FUNCTION_BLOCK PlantProcess
  (* Standard: 61499-2 *)
  (* Version 0.1, 2017-00-02, hpea485, UOA *)
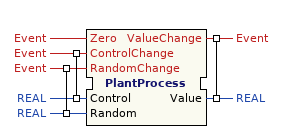
  EVENT_INPUT
    Zero;
    ControlChange WITH Control;
    RandomChange WITH Random;
  END_EVENT
  EVENT_OUTPUT
    ValueChange WITH Value;
  END_EVENT
  VAR_INPUT
    Control : REAL;
    Random : REAL := 0.0;
  END_VAR
  VAR_OUTPUT
    Value : REAL;
  END_VAR
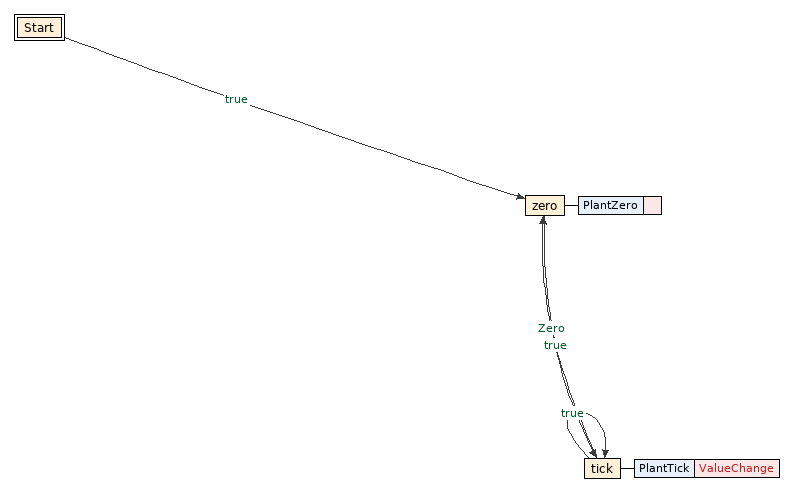
  EC_STATES
    Start;
    zero : PlantZero;
    tick : PlantTick -> ValueChange;
  END_STATES
  EC_TRANSITIONS
    Start TO zero := true;
    zero TO tick := true;
    tick TO zero := Zero;
    tick TO tick := true;
  END_TRANSITIONS
  ALGORITHM PlantZero IN C:
me->Value = 0;
  END_ALGORITHM
  ALGORITHM PlantTick IN C:
me->Value += me->Control + me->Random;
  END_ALGORITHM
END_FUNCTION_BLOCK
